FUNCTION fnKonwersja2x16naFloat32BySchneider : BOOL
  VAR_INPUT
    wRejestrMSW : WORD;  (* MSW - Most Significant Word *)
    wRejestrLSW : WORD;  (* LSW - Least Significant Word *)
  END_VAR
  VAR_IN_OUT
    rWartoscFloat32 : REAL;
  END_VAR
  VAR
    rZnak : REAL;
    rTempMSW : REAL;
    rTempMSW2 : REAL;
    wTempMSW : WORD;
    wTempMSW2 : WORD;
    dwTemp : DWORD;
    lrStala1 : LREAL := 8388608.0;
    lrStala2 : LREAL := 4194304.0;
    lrTemp : LREAL;
    rFaction : REAL;
    rExponent : REAL;
  END_VAR

            (*			
Autor:					Paweł Kąkol, 
Prawa majątkowe: 		Solwena Sp. z o.o., 
Aktualizacje:			2017-11-03-13:45-PK

Opis:					Funkcja do konwersji 2 rejestrów modbusowych na zmienną Float32 by Schneider Electric
*)
wTempMSW := wRejestrMSW / 256; // wyciagniecie 8 starszych bitow
//ustalanie znaku
IF (wTempMSW AND 128) = 128 THEN
	rZnak := -1.0;
	wTempMSW := wTempMSW AND 127; // usuniecie bitu znaku
ELSE
	rZnak := 1.0;
END_IF
wTempMSW2 := wRejestrMSW MOD 256; // wyciagniecie 8 mlodszych bitow
wTempMSW := (wTempMSW * 2) + ((wTempMSW2 AND 128) / 128); //przesuniecie bitowe o 1 w lewo wraz z dodaniem na najmlodsza pozycje najstarszego bitu z młodszych 8 bitow
wTempMSW2 := wTempMSW2 AND 127;// usuniecie najstarszego bitu
rExponent := WORD_TO_REAL(wTempMSW) - 127.0; // wyznaczanie wykladnika
dwTemp := WORD_TO_DWORD(wTempMSW2); //konwersja zmiennej 16-bitowej na 32-bitowa
dwTemp := dwTemp * 65536; //przesuniecie bitowe w lewo o 16 pozycji
dwTemp := dwTemp + WORD_TO_DWORD(wRejestrLSW); // dostawienie na koncu 16 bitow zmiennej LSW
lrTemp := DWORD_TO_LREAL(dwTemp);
//wybieranie ulamka
IF wTempMSW > 0 THEN
	rFaction := LREAL_TO_REAL((lrTemp / lrStala1) + 1.0);
ELSE
	rFaction := LREAL_TO_REAL(lrTemp / lrStala2);
END_IF
//obliczanie wartosci Float32
rWartoscFloat32 := rZnak * rFaction * EXPT(2.0, rExponent);
          
END_FUNCTION

FUNCTION fnKonwersja4x128na512 : BOOL
  VAR_INPUT
    sKomunikatCzesc1 : STRING(128);
    sKomunikatCzesc2 : STRING(128);
    sKomunikatCzesc3 : STRING(128);
    sKomunikatCzesc4 : STRING(128);
  END_VAR
  VAR_IN_OUT
    sKomunikat512 : alSTRINGKomunikat;
  END_VAR

            sKomunikat512 := CONCAT(sKomunikatCzesc1 , sKomunikatCzesc2);
sKomunikat512 := CONCAT(sKomunikat512 , sKomunikatCzesc3);
sKomunikat512 := CONCAT(sKomunikat512 , sKomunikatCzesc4);
          
END_FUNCTION

FUNCTION fnKonwersja512na4x128 : BOOL
  VAR_INPUT
    sKomunikat512 : alSTRINGKomunikat;
  END_VAR
  VAR_IN_OUT
    sKomunikatCzesc1 : STRING(128);
    sKomunikatCzesc2 : STRING(128);
    sKomunikatCzesc3 : STRING(128);
    sKomunikatCzesc4 : STRING(128);
  END_VAR

            sKomunikatCzesc1 := MID(sKomunikat512 , 128 , 1);
sKomunikatCzesc2 := MID(sKomunikat512 , 128 , 129);
sKomunikatCzesc3 := MID(sKomunikat512 , 128 , 513);
sKomunikatCzesc4 := MID(sKomunikat512 , 128 , 385);
fnKonwersja512na4x128 := TRUE;

          
END_FUNCTION

FUNCTION fnKonwersjaDEC_BYTE_TO_HEX_STRING : STRING(2)
  VAR_INPUT
    bWartoscDEC : BYTE;
  END_VAR
  VAR CONSTANT
    sTablicaReprezentacjiHEX : ARRAY[0..255] OF STRING(2) := ['00', '01', '02', '03', '04', '05', '06', '07', '08', '09', '0A', '0B', '0C', '0D', '0E', '0F', '10', '11', '12', '13', '14', '15', '16', '17', '18', '19', '1A', '1B', '1C', '1D', '1E', '1F', '20', '21', '22', '23', '24', '25', '26', '27', '28', '29', '2A', '2B', '2C', '2D', '2E', '2F', '30', '31', '32', '33', '34', '35', '36', '37', '38', '39', '3A', '3B', '3C', '3D', '3E', '3F', '40', '41', '42', '43', '44', '45', '46', '47', '48', '49', '4A', '4B', '4C', '4D', '4E', '4F', '50', '51', '52', '53', '54', '55', '56', '57', '58', '59', '5A', '5B', '5C', '5D', '5E', '5F', '60', '61', '62', '63', '64', '65', '66', '67', '68', '69', '6A', '6B', '6C', '6D', '6E', '6F', '70', '71', '72', '73', '74', '75', '76', '77', '78', '79', '7A', '7B', '7C', '7D', '7E', '7F', '80', '81', '82', '83', '84', '85', '86', '87', '88', '89', '8A', '8B', '8C', '8D', '8E', '8F', '90', '91', '92', '93', '94', '95', '96', '97', '98', '99', '9A', '9B', '9C', '9D', '9E', '9F', 'A0', 'A1', 'A2', 'A3', 'A4', 'A5', 'A6', 'A7', 'A8', 'A9', 'AA', 'AB', 'AC', 'AD', 'AE', 'AF', 'B0', 'B1', 'B2', 'B3', 'B4', 'B5', 'B6', 'B7', 'B8', 'B9', 'BA', 'BB', 'BC', 'BD', 'BE', 'BF', 'C0', 'C1', 'C2', 'C3', 'C4', 'C5', 'C6', 'C7', 'C8', 'C9', 'CA', 'CB', 'CC', 'CD', 'CE', 'CF', 'D0', 'D1', 'D2', 'D3', 'D4', 'D5', 'D6', 'D7', 'D8', 'D9', 'DA', 'DB', 'DC', 'DD', 'DE', 'DF', 'E0', 'E1', 'E2', 'E3', 'E4', 'E5', 'E6', 'E7', 'E8', 'E9', 'EA', 'EB', 'EC', 'ED', 'EE', 'EF', 'F0', 'F1', 'F2', 'F3', 'F4', 'F5', 'F6', 'F7', 'F8', 'F9', 'FA', 'FB', 'FC', 'FD', 'FE', 'FF'];
  END_VAR

            (*			
Autor:					Paweł Kąkol, 
Prawa majątkowe: 		Solwena Sp. z o.o., 
Aktualizacje:			2018-08-24-PK - stworzenie

Opis:					Funkcja zwraca reprezentację szesnastkową w Stringu wartości dziesiętnej podanej jako BYTE;
*)

fnKonwersjaDEC_BYTE_TO_HEX_STRING := sTablicaReprezentacjiHEX[bWartoscDEC];
          
END_FUNCTION

FUNCTION fnKonwersjaHEX_STRING_TO_DEC_BYTE : BYTE
  VAR_INPUT
    sWartoscHEX : STRING(2);
  END_VAR
  VAR CONSTANT
    sTablicaReprezentacjiHEX : ARRAY[0..15] OF STRING(1) := ['0', '1', '2', '3', '4', '5', '6', '7', '8', '9', 'A', 'B', 'C', 'D', 'E', 'F'];
  END_VAR
  VAR
    sPierwszyZnak : STRING(1);
    sDrugiZnak : STRING(1);
    bPetla : BYTE;
  END_VAR

            (*			
Autor:					Paweł Kąkol, 
Prawa majątkowe: 		Solwena Sp. z o.o., 
Aktualizacje:			2018-08-24-PK - stworzenie

Opis:					Funkcja zwraca reprezentację dziesiętną jako BYTE wartości szesnastkowej podanej jako STRING;
*)

sPierwszyZnak := LEFT(sWartoscHEX, 1);
FOR bPetla := 0 TO 15 BY 1 DO
	IF sPierwszyZnak = sTablicaReprezentacjiHEX[bPetla] THEN
		fnKonwersjaHEX_STRING_TO_DEC_BYTE := bPetla * 16;
	END_IF
END_FOR
sDrugiZnak := RIGHT(sWartoscHEX, 1);
FOR bPetla := 0 TO 15 BY 1 DO
	IF sDrugiZnak = sTablicaReprezentacjiHEX[bPetla] THEN
		fnKonwersjaHEX_STRING_TO_DEC_BYTE := fnKonwersjaHEX_STRING_TO_DEC_BYTE + bPetla;
	END_IF
END_FOR

          
END_FUNCTION

FUNCTION fnKonwersjaINT_STRING : STRING
  VAR_INPUT
    intWartosc : INT;
    intIloscZnakow : INT;
  END_VAR

            fnKonwersjaINT_STRING := INT_TO_STRING(intWartosc);

IF intWartosc < 100000 AND intIloscZnakow > 5 THEN
	fnKonwersjaINT_STRING := CONCAT('0' , fnKonwersjaINT_STRING);
END_IF

IF intWartosc < 10000 AND intIloscZnakow > 4 THEN
	fnKonwersjaINT_STRING := CONCAT('0' , fnKonwersjaINT_STRING);
END_IF

IF intWartosc < 1000 AND intIloscZnakow > 3 THEN
	fnKonwersjaINT_STRING := CONCAT('0' , fnKonwersjaINT_STRING);
END_IF

IF intWartosc < 100 AND intIloscZnakow > 2 THEN
	fnKonwersjaINT_STRING := CONCAT('0' , fnKonwersjaINT_STRING);
END_IF

IF intWartosc < 10 AND intIloscZnakow > 1 THEN
	fnKonwersjaINT_STRING := CONCAT('0' , fnKonwersjaINT_STRING);
END_IF

          
END_FUNCTION

FUNCTION fnModbusZapisRejestru : BOOL
  VAR_INPUT
    bAdresUrzadzenia : BYTE;  (* ID urządzenia SLAVE w sieci MODBUS *)
    bFunkcja : BYTE;  (* kod funkcji użytej w rozkazie MODBUS *)
    uiAdresRejestru : UINT;  (* rejestr startowy *)
    pZmiennaReferencyjna : POINTER TO WORD;  (* wskaźnik do wartości do zapisu *)
    wWartoscDoZapisania : WORD;  (* wartość do zapisania *)
    intModbusOdczytZapisZadanieRozmiar : INT;
  END_VAR
  VAR_IN_OUT
    arModbusOdczytZapisZadanie : ARRAY[1..1000] OF typModbusOdczytZapisZadanie;
    intModbusOdczytZapisZadanieZnacznikZapisu : INT;
  END_VAR

            fnTablicaKomunikatowInkrementacja(intRozmiarTablicy := intModbusOdczytZapisZadanieRozmiar , intWskaznik := intModbusOdczytZapisZadanieZnacznikZapisu);

arModbusOdczytZapisZadanie[intModbusOdczytZapisZadanieZnacznikZapisu].bAdresUrzadzenia := bAdresUrzadzenia;
arModbusOdczytZapisZadanie[intModbusOdczytZapisZadanieZnacznikZapisu].bFunkcja := bFunkcja;
arModbusOdczytZapisZadanie[intModbusOdczytZapisZadanieZnacznikZapisu].uiAdresRejestru := uiAdresRejestru;
arModbusOdczytZapisZadanie[intModbusOdczytZapisZadanieZnacznikZapisu].pZmiennaDoOdczytu := pZmiennaReferencyjna;
arModbusOdczytZapisZadanie[intModbusOdczytZapisZadanieZnacznikZapisu].wWartoscDoZapisania := wWartoscDoZapisania;
          
END_FUNCTION

FUNCTION fnOdwrocenieBitowTemperaturyUjemnejREAL_TO_WORD : WORD
  VAR_INPUT
    rTemperaturaKelviny : REAL;
  END_VAR

            (*			
Autor:					Artur Wyszomirski, 2019-05-27 
Prawa majątkowe: 		Solwena Sp. z o.o., 
Aktualizacje:			 
					
Opis:					Funkcja odwraca bity temperatury, jeśli tempratura jest mniejsza ujemna w skali Celsjusza. Wartość wejściowa w REAL, wartość wyjściowa w WORD.
*)
IF rTemperaturaKelviny < 273.15 THEN	// Jeśli temperatura jest ujemna, odwróć bity
	fnOdwrocenieBitowTemperaturyUjemnejREAL_TO_WORD := REAL_TO_WORD(65535 - (ABS(rTemperaturaKelviny - 273.15) * 10));	
ELSE
	fnOdwrocenieBitowTemperaturyUjemnejREAL_TO_WORD := REAL_TO_WORD((rTemperaturaKelviny - 273.15) * 10);						
END_IF
          
END_FUNCTION

FUNCTION fnRozbicieNaBityRejestru16Bit : BOOL
  VAR_INPUT
    wRejestr16Bit : WORD;
  END_VAR
  VAR_OUTPUT
    xBit0 : BOOL;
    xBit1 : BOOL;
    xBit2 : BOOL;
    xBit3 : BOOL;
    xBit4 : BOOL;
    xBit5 : BOOL;
    xBit6 : BOOL;
    xBit7 : BOOL;
    xBit8 : BOOL;
    xBit9 : BOOL;
    xBit10 : BOOL;
    xBit11 : BOOL;
    xBit12 : BOOL;
    xBit13 : BOOL;
    xBit14 : BOOL;
    xBit15 : BOOL;
  END_VAR
  VAR
    wTempRejestr16 : WORD;
  END_VAR

            (*			
Autor:					Paweł Kąkol, 
Prawa majątkowe: 		Solwena Sp. z o.o., 
Aktualizacje:			2017-11-17-10:00-PK

Opis:					Funkcja do rozbijania rejestru 16-bitowego typu WORD na pojedyncze zmienne BOOL,
						Nalezy pamietac, ze numeracja bitow jest zgodna z odpowiadajacymi wykladnikami potegi liczby 2
*)
wTempRejestr16 := wRejestr16Bit;
//sprawdzanie stanu bitow
IF wTempRejestr16 >= 32768 THEN
	xBit15 := TRUE;
	wTempRejestr16 := wTempRejestr16 MOD 32768;
ELSE
	xBit15 := FALSE;	
END_IF
IF wTempRejestr16 >= 16384 THEN
	xBit14 := TRUE;
	wTempRejestr16 := wTempRejestr16 MOD 16384;
ELSE
	xBit14 := FALSE;
END_IF
IF wTempRejestr16 >= 8192 THEN
	xBit13 := TRUE;
	wTempRejestr16 := wTempRejestr16 MOD 8192;
ELSE
	xBit13 := FALSE;
END_IF
IF wTempRejestr16 >= 4096 THEN
	xBit12 := TRUE;
	wTempRejestr16 := wTempRejestr16 MOD 4096;
ELSE
	xBit12 := FALSE;
END_IF
IF wTempRejestr16 >= 2048 THEN
	xBit11 := TRUE;
	wTempRejestr16 := wTempRejestr16 MOD 2048;
ELSE
	xBit11 := FALSE;
END_IF
IF wTempRejestr16 >= 1024 THEN
	xBit10 := TRUE;
	wTempRejestr16 := wTempRejestr16 MOD 1024;
ELSE
	xBit10 := FALSE;
END_IF
IF wTempRejestr16 >= 512 THEN
	xBit9 := TRUE;
	wTempRejestr16 := wTempRejestr16 MOD 512;
ELSE
	xBit9 := FALSE;
END_IF
IF wTempRejestr16 >= 256 THEN
	xBit8 := TRUE;
	wTempRejestr16 := wTempRejestr16 MOD 256;
ELSE
	xBit8 := FALSE;
END_IF
IF wTempRejestr16 >= 128 THEN
	xBit7 := TRUE;
	wTempRejestr16 := wTempRejestr16 MOD 128;
ELSE
	xBit7 := FALSE;
END_IF
IF wTempRejestr16 >= 64 THEN
	xBit6 := TRUE;
	wTempRejestr16 := wTempRejestr16 MOD 64;
ELSE
	xBit6 := FALSE;
END_IF
IF wTempRejestr16 >= 32 THEN
	xBit5 := TRUE;
	wTempRejestr16 := wTempRejestr16 MOD 32;
ELSE
	xBit5 := FALSE;
END_IF
IF wTempRejestr16 >= 16 THEN
	xBit4 := TRUE;
	wTempRejestr16 := wTempRejestr16 MOD 16;
ELSE
	xBit4 := FALSE;
END_IF
IF wTempRejestr16 >= 8 THEN
	xBit3 := TRUE;
	wTempRejestr16 := wTempRejestr16 MOD 8;
ELSE
	xBit3 := FALSE;
END_IF
IF wTempRejestr16 >= 4 THEN
	xBit2 := TRUE;
	wTempRejestr16 := wTempRejestr16 MOD 4;
ELSE
	xBit2 := FALSE;
END_IF
IF wTempRejestr16 >= 2 THEN
	xBit1 := TRUE;
	wTempRejestr16 := wTempRejestr16 MOD 2;
ELSE
	xBit1 := FALSE;
END_IF
IF wTempRejestr16 >= 1 THEN
	xBit0 := TRUE;
ELSE
	xBit0 := FALSE;
END_IF
          
END_FUNCTION

FUNCTION fnTablicaKomunikatowInkrementacja : BOOL
  VAR_INPUT
    intRozmiarTablicy : INT;
  END_VAR
  VAR_IN_OUT
    intWskaznik : INT;
  END_VAR

            intWskaznik := 	intWskaznik + 1; 
IF intWskaznik > intRozmiarTablicy THEN
	intWskaznik := 1;
END_IF

          
END_FUNCTION

FUNCTION fnZapiszKomunikat : BOOL
  VAR_INPUT
    sCalyKomunikat : alSTRINGKomunikat;
    sTypKomunikatu : STRING;
    sMnemonik : STRING;
    sMACAdres : STRING;
    sIdNadawcy : STRING;
    sIdOdbiorcy : STRING;
    sDaneZapasowe : STRING;
    sDane : alSTRINGKomunikat;
    intTablicaKomunikatowRozmiar : INT;
  END_VAR
  VAR_IN_OUT
    intTablicaKomunikatowZnacznikZapisu : INT;
    arTablicaKomunikatow : alARRAYTablicaKomunikatow;
    sWyslanyKomunikat : alSTRINGKomunikat;
  END_VAR
  VAR
    sKomunikat : alSTRINGKomunikat;
    intBlad : INT;
    typKomunikat : typKomunikat;
  END_VAR

            (* blok do zapisu nowego komunikatu w buforze do wysłania*)

IF sCalyKomunikat = '' THEN
	typKomunikat.sZnacznik := 'ˆ';
	typKomunikat.sTypKomunikatu := sTypKomunikatu;
	typKomunikat.sMnemonikWlasciciela := LEFT(sMnemonik , 3);
	typKomunikat.sMnemonikWlascicielaExt := Right(sMnemonik , 1);
	typKomunikat.sMACAdres := sMACAdres;
	typKomunikat.sIDZrodla := sIdNadawcy;
	typKomunikat.sIDPrzeznaczenia := sIdOdbiorcy;
	typKomunikat.sRezerwa := sDaneZapasowe;
	typKomunikat.sDane := sDane;
	fnKomunikatInOut(	xStringNaStrukture := FALSE ,
						xStringUpdateZeStruktury := FALSE ,
						xStrukturyNaString := TRUE ,
						xWyczyscStrukture := FALSE ,
						xAktualizujZnacznikCzasu := TRUE ,
						xAktualizujDlugoscDanych := TRUE ,
						sKomunikat := sKomunikat ,
						typKomunikat := typKomunikat ,
						intBlad := intBlad);
	ELSE
	sKomunikat := sCalyKomunikat;
END_IF
fnTablicaKomunikatowInkrementacja(intWskaznik := intTablicaKomunikatowZnacznikZapisu , intRozmiarTablicy := intTablicaKomunikatowRozmiar);
arTablicaKomunikatow[intTablicaKomunikatowZnacznikZapisu] := sKomunikat;
sWyslanyKomunikat := sKomunikat;

          
END_FUNCTION

FUNCTION fnZlozenieBitowWRejestr16Bit : BOOL
  VAR_INPUT
    xBit0 : BOOL;
    xBit1 : BOOL;
    xBit2 : BOOL;
    xBit3 : BOOL;
    xBit4 : BOOL;
    xBit5 : BOOL;
    xBit6 : BOOL;
    xBit7 : BOOL;
    xBit8 : BOOL;
    xBit9 : BOOL;
    xBit10 : BOOL;
    xBit11 : BOOL;
    xBit12 : BOOL;
    xBit13 : BOOL;
    xBit14 : BOOL;
    xBit15 : BOOL;
  END_VAR
  VAR_OUTPUT
    wRejestr16Bit : WORD;
  END_VAR

            (*			
Autor:					Paweł Kąkol, 
Prawa majątkowe: 		Solwena Sp. z o.o., 
Aktualizacje:			2017-12-13-09:30-PK - stworzenie

Opis:					Funkcja do składania rejestru 16-bitowego typu WORD z pojedynczych zmiennych BOOL,
						Nalezy pamietac, ze numeracja bitow jest zgodna z odpowiadajacymi wykladnikami potegi liczby 2
*)
wRejestr16Bit := 0;
//sprawdzanie stanu bitow
IF xBit0 THEN
	wRejestr16Bit := 1;	
END_IF
IF xBit1 THEN
	wRejestr16Bit := wRejestr16Bit + 2;	
END_IF
IF xBit1 THEN
	wRejestr16Bit := wRejestr16Bit + 4;	
END_IF
IF xBit1 THEN
	wRejestr16Bit := wRejestr16Bit + 8;	
END_IF
IF xBit1 THEN
	wRejestr16Bit := wRejestr16Bit + 16;	
END_IF
IF xBit1 THEN
	wRejestr16Bit := wRejestr16Bit + 32;	
END_IF
IF xBit1 THEN
	wRejestr16Bit := wRejestr16Bit + 64;	
END_IF
IF xBit1 THEN
	wRejestr16Bit := wRejestr16Bit + 128;	
END_IF
IF xBit1 THEN
	wRejestr16Bit := wRejestr16Bit + 256;	
END_IF
IF xBit1 THEN
	wRejestr16Bit := wRejestr16Bit + 512;	
END_IF
IF xBit1 THEN
	wRejestr16Bit := wRejestr16Bit + 1024;	
END_IF
IF xBit1 THEN
	wRejestr16Bit := wRejestr16Bit + 2048;	
END_IF
IF xBit1 THEN
	wRejestr16Bit := wRejestr16Bit + 4096;	
END_IF
IF xBit1 THEN
	wRejestr16Bit := wRejestr16Bit + 8192;	
END_IF
IF xBit1 THEN
	wRejestr16Bit := wRejestr16Bit + 16384;	
END_IF
IF xBit1 THEN
	wRejestr16Bit := wRejestr16Bit + 32768;	
END_IF
          
END_FUNCTION
